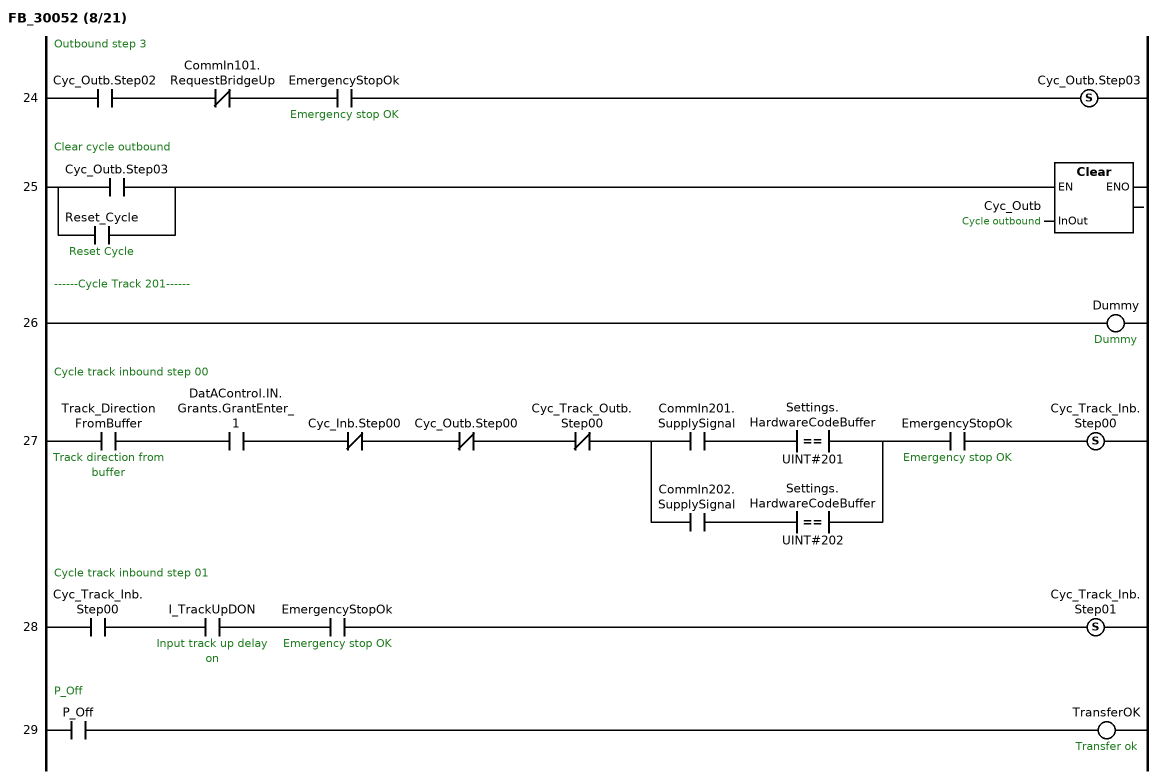
(* [picture p246: FB_30052, rungs 24-29] *)
(* Rung 24: Outbound step 3 *)
IF Cyc_Outb.Step02 AND NOT CommIn101.RequestBridgeUp AND EmergencyStopOk THEN
    Cyc_Outb.Step03 := TRUE;
END_IF;
(* Rung 25: Clear cycle outbound *)
IF Cyc_Outb.Step03 OR Reset_Cycle THEN Clear(InOut := Cyc_Outb); END_IF;
(* Rung 26: ------Cycle Track 201------ *)
Dummy := TRUE;
(* Rung 27: Cycle track inbound step 00 *)
IF Track_DirectionFromBuffer AND DatAControl.IN.Grants.GrantEnter_1 AND NOT Cyc_Inb.Step00 AND NOT Cyc_Outb.Step00 AND NOT Cyc_Track_Outb.Step00 AND ((CommIn201.SupplySignal AND (Settings.HardwareCodeBuffer = UINT#201)) OR (CommIn202.SupplySignal AND (Settings.HardwareCodeBuffer = UINT#202))) AND EmergencyStopOk THEN
    Cyc_Track_Inb.Step00 := TRUE;
END_IF;
(* Rung 28: Cycle track inbound step 01 *)
IF Cyc_Track_Inb.Step00 AND I_TrackUpDON AND EmergencyStopOk THEN Cyc_Track_Inb.Step01 := TRUE; END_IF;
(* Rung 29: P_Off *)
TransferOK := P_Off;

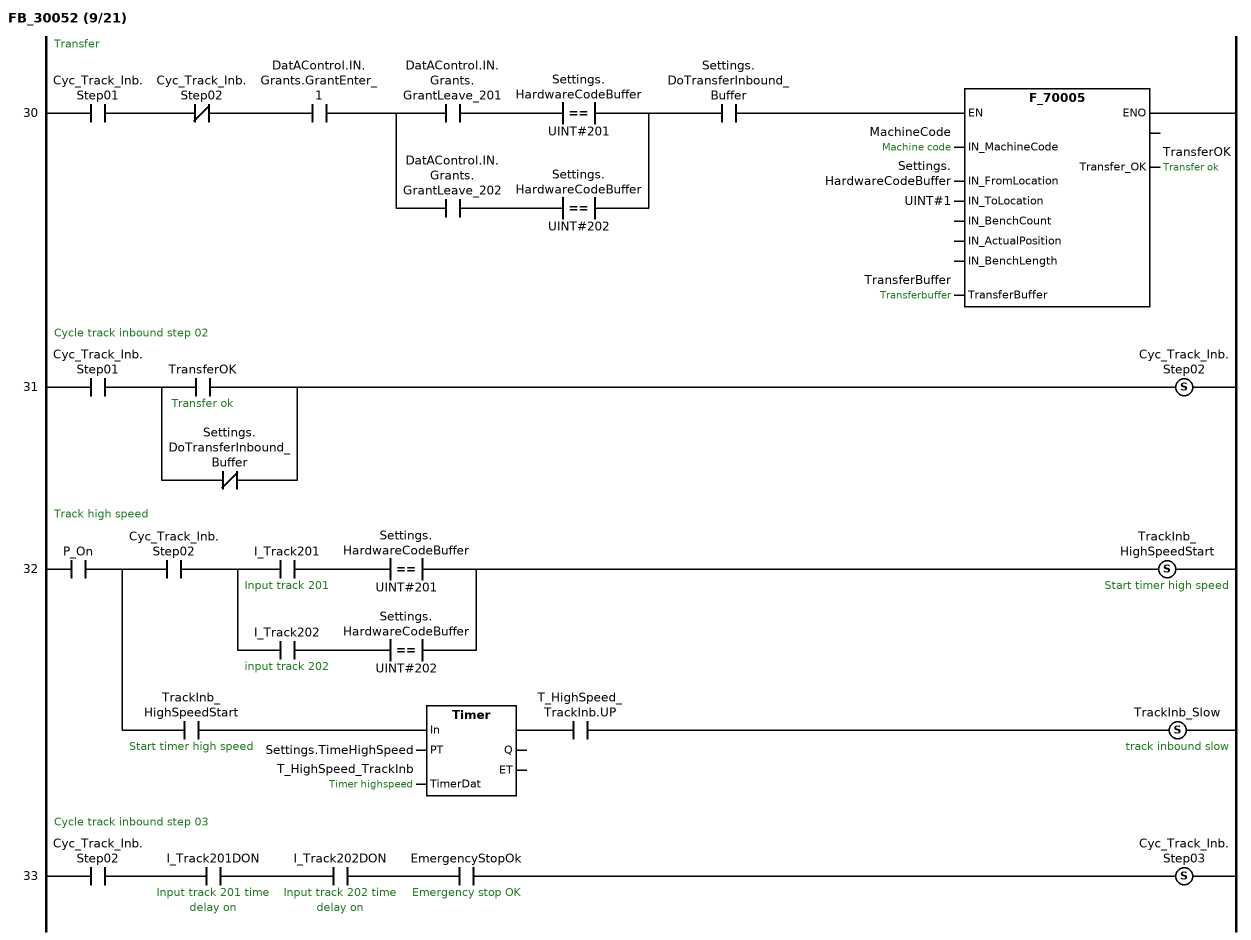
(* Rung 30: Transfer *)
IF Cyc_Track_Inb.Step01 AND NOT Cyc_Track_Inb.Step02 AND DatAControl.IN.Grants.GrantEnter_1 AND ((DatAControl.IN.Grants.GrantLeave_201 AND (Settings.HardwareCodeBuffer = UINT#201)) OR (DatAControl.IN.Grants.GrantLeave_202 AND (Settings.HardwareCodeBuffer = UINT#202))) AND Settings.DoTransferInbound_Buffer THEN
    F_70005(IN_MachineCode := MachineCode, IN_FromLocation := Settings.HardwareCodeBuffer, IN_ToLocation := UINT#1, TransferBuffer := TransferBuffer, Transfer_OK => TransferOK);
END_IF;
(* Rung 31: Cycle track inbound step 02 *)
IF Cyc_Track_Inb.Step01 AND (TransferOK OR NOT Settings.DoTransferInbound_Buffer) THEN
    Cyc_Track_Inb.Step02 := TRUE;
END_IF;
(* Rung 32: Track high speed *)
IF P_On AND Cyc_Track_Inb.Step02 AND ((I_Track201 AND (Settings.HardwareCodeBuffer = UINT#201)) OR (I_Track202 AND (Settings.HardwareCodeBuffer = UINT#202))) THEN
    TrackInb_HighSpeedStart := TRUE;
END_IF;
_t2 := Timer(In := P_On AND TrackInb_HighSpeedStart, PT := Settings.TimeHighSpeed, TimerDat := T_HighSpeed_TrackInb);
IF _t2 AND T_HighSpeed_TrackInb.UP THEN TrackInb_Slow := TRUE; END_IF;
(* Rung 33: Cycle track inbound step 03 *)
IF Cyc_Track_Inb.Step02 AND I_Track201DON AND I_Track202DON AND EmergencyStopOk THEN
    Cyc_Track_Inb.Step03 := TRUE;
END_IF;

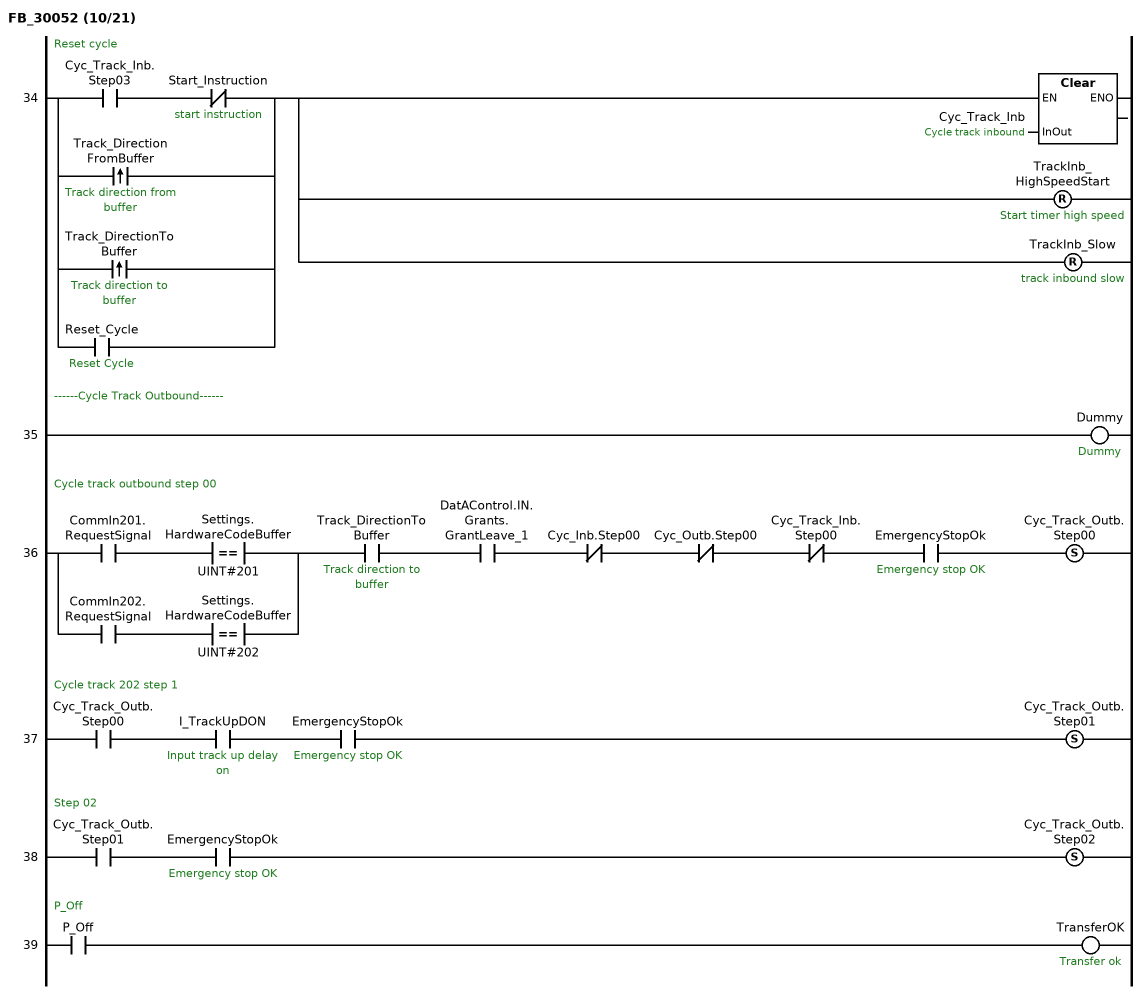
(* Rung 34: Reset cycle *)
_e3(CLK := Track_DirectionFromBuffer);
_e4(CLK := Track_DirectionToBuffer);
_p5 := (Cyc_Track_Inb.Step03 AND NOT Start_Instruction) OR _e3.Q OR _e4.Q OR Reset_Cycle;
IF _p5 THEN
    Clear(InOut := Cyc_Track_Inb);
    TrackInb_HighSpeedStart := FALSE;
    TrackInb_Slow := FALSE;
END_IF;
(* Rung 35: ------Cycle Track Outbound------ *)
Dummy := TRUE;
(* Rung 36: Cycle track outbound step 00 *)
IF ((CommIn201.RequestSignal AND (Settings.HardwareCodeBuffer = UINT#201)) OR (CommIn202.RequestSignal AND (Settings.HardwareCodeBuffer = UINT#202))) AND Track_DirectionToBuffer AND DatAControl.IN.Grants.GrantLeave_1 AND NOT Cyc_Inb.Step00 AND NOT Cyc_Outb.Step00 AND NOT Cyc_Track_Inb.Step00 AND EmergencyStopOk THEN
    Cyc_Track_Outb.Step00 := TRUE;
END_IF;
(* Rung 37: Cycle track 202 step 1 *)
IF Cyc_Track_Outb.Step00 AND I_TrackUpDON AND EmergencyStopOk THEN Cyc_Track_Outb.Step01 := TRUE; END_IF;
(* Rung 38: Step 02 *)
IF Cyc_Track_Outb.Step01 AND EmergencyStopOk THEN Cyc_Track_Outb.Step02 := TRUE; END_IF;
(* Rung 39: P_Off *)
TransferOK := P_Off;

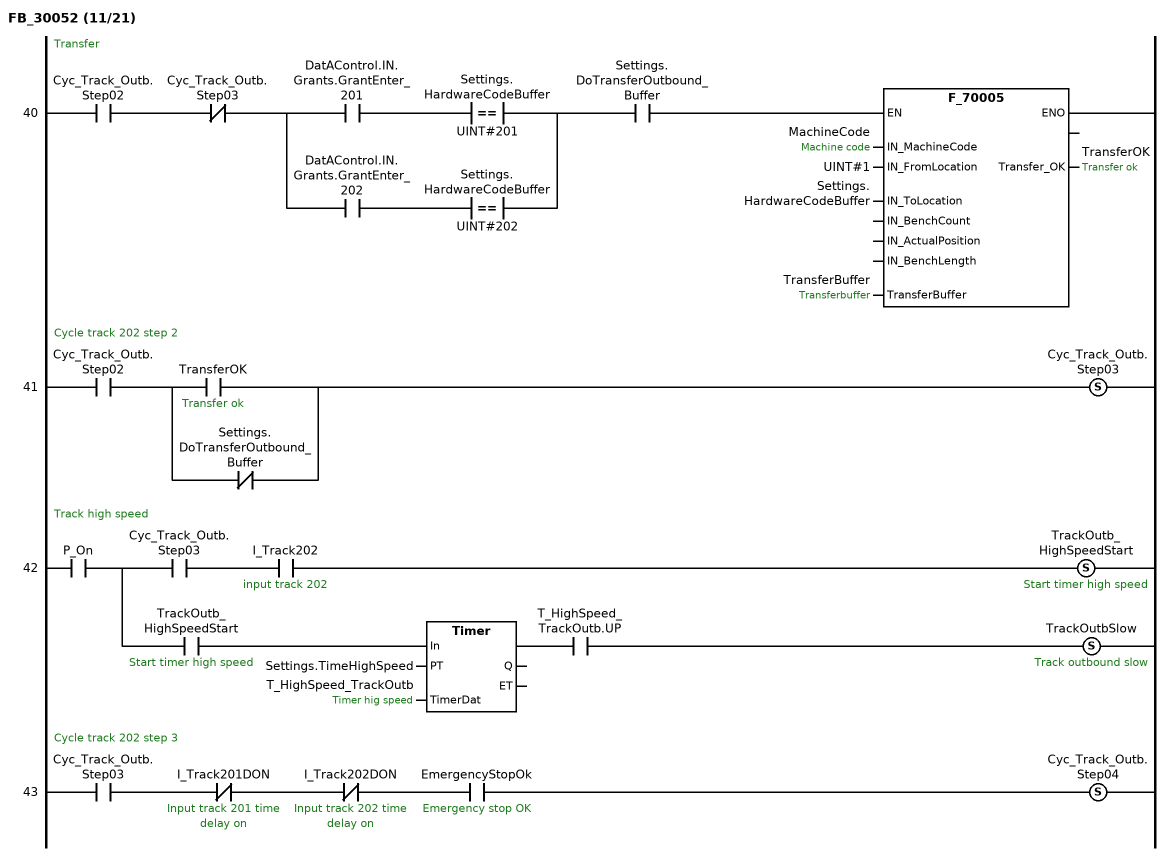
(* Rung 40: Transfer *)
IF Cyc_Track_Outb.Step02 AND NOT Cyc_Track_Outb.Step03 AND ((DatAControl.IN.Grants.GrantEnter_201 AND (Settings.HardwareCodeBuffer = UINT#201)) OR (DatAControl.IN.Grants.GrantEnter_202 AND (Settings.HardwareCodeBuffer = UINT#202))) AND Settings.DoTransferOutbound_Buffer THEN
    F_70005(IN_MachineCode := MachineCode, IN_FromLocation := UINT#1, IN_ToLocation := Settings.HardwareCodeBuffer, TransferBuffer := TransferBuffer, Transfer_OK => TransferOK);
END_IF;
(* Rung 41: Cycle track 202 step 2 *)
IF Cyc_Track_Outb.Step02 AND (TransferOK OR NOT Settings.DoTransferOutbound_Buffer) THEN
    Cyc_Track_Outb.Step03 := TRUE;
END_IF;
(* Rung 42: Track high speed *)
IF P_On AND Cyc_Track_Outb.Step03 AND I_Track202 THEN TrackOutb_HighSpeedStart := TRUE; END_IF;
_t6 := Timer(In := P_On AND TrackOutb_HighSpeedStart, PT := Settings.TimeHighSpeed, TimerDat := T_HighSpeed_TrackOutb);
IF _t6 AND T_HighSpeed_TrackOutb.UP THEN TrackOutbSlow := TRUE; END_IF;
(* Rung 43: Cycle track 202 step 3 *)
IF Cyc_Track_Outb.Step03 AND NOT I_Track201DON AND NOT I_Track202DON AND EmergencyStopOk THEN
    Cyc_Track_Outb.Step04 := TRUE;
END_IF;

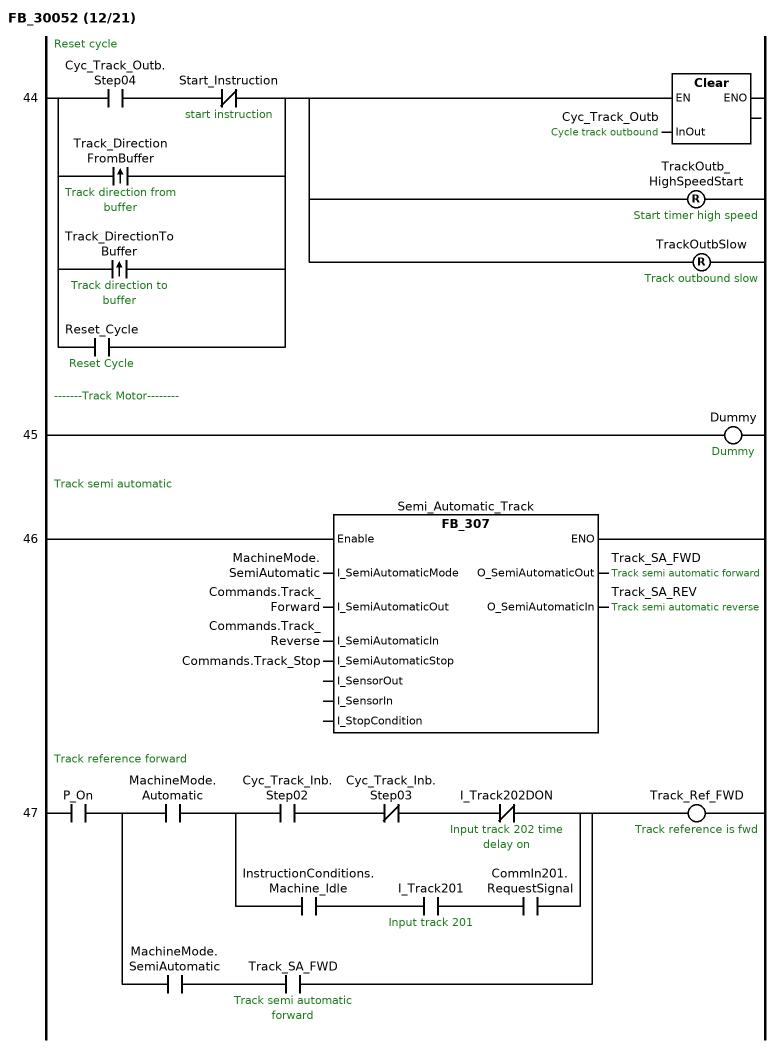
(* Rung 44: Reset cycle *)
_e7(CLK := Track_DirectionFromBuffer);
_e8(CLK := Track_DirectionToBuffer);
_p9 := (Cyc_Track_Outb.Step04 AND NOT Start_Instruction) OR _e7.Q OR _e8.Q OR Reset_Cycle;
IF _p9 THEN
    Clear(InOut := Cyc_Track_Outb);
    TrackOutb_HighSpeedStart := FALSE;
    TrackOutbSlow := FALSE;
END_IF;
(* Rung 45: -------Track Motor-------- *)
Dummy := TRUE;
(* Rung 46: Track semi automatic *)
Semi_Automatic_Track(Enable := TRUE, I_SemiAutomaticMode := MachineMode.SemiAutomatic, I_SemiAutomaticOut := Commands.Track_Forward, I_SemiAutomaticIn := Commands.Track_Reverse, I_SemiAutomaticStop := Commands.Track_Stop, O_SemiAutomaticOut => Track_SA_FWD, O_SemiAutomaticIn => Track_SA_REV);
(* Rung 47: Track reference forward *)
Track_Ref_FWD := P_On AND ((MachineMode.Automatic AND ((Cyc_Track_Inb.Step02 AND NOT Cyc_Track_Inb.Step03 AND NOT I_Track202DON) OR (InstructionConditions.Machine_Idle AND I_Track201 AND CommIn201.RequestSignal))) OR (MachineMode.SemiAutomatic AND Track_SA_FWD));

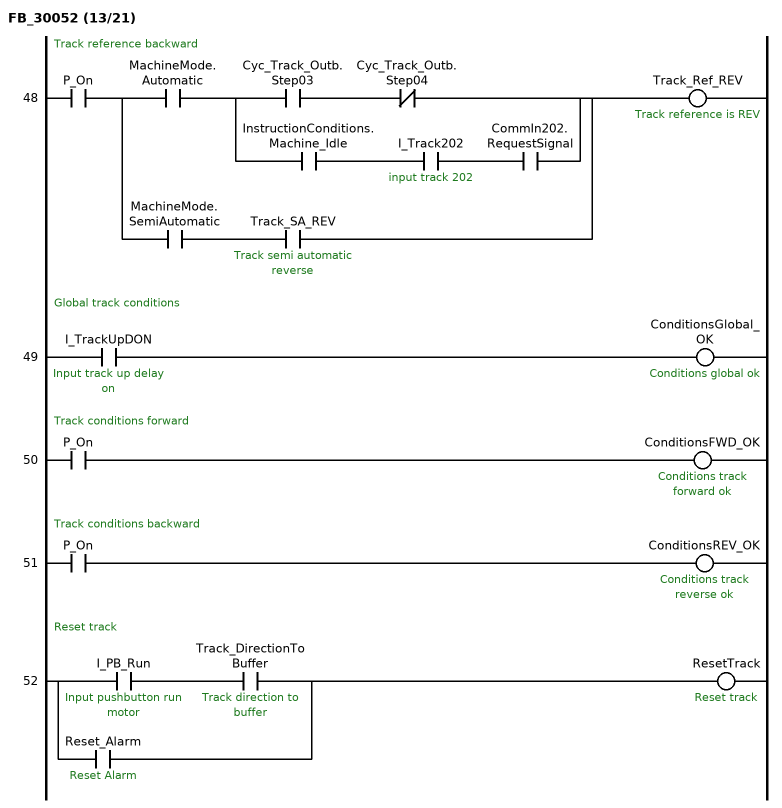
(* Rung 48: Track reference backward *)
Track_Ref_REV := P_On AND ((MachineMode.Automatic AND ((Cyc_Track_Outb.Step03 AND NOT Cyc_Track_Outb.Step04) OR (InstructionConditions.Machine_Idle AND I_Track202 AND CommIn202.RequestSignal))) OR (MachineMode.SemiAutomatic AND Track_SA_REV));
(* Rung 49: Global track conditions *)
ConditionsGlobal_OK := I_TrackUpDON;
(* Rung 50: Track conditions forward *)
ConditionsFWD_OK := P_On;
(* Rung 51: Track conditions backward *)
ConditionsREV_OK := P_On;
(* Rung 52: Reset track *)
ResetTrack := (I_PB_Run AND Track_DirectionToBuffer) OR Reset_Alarm;

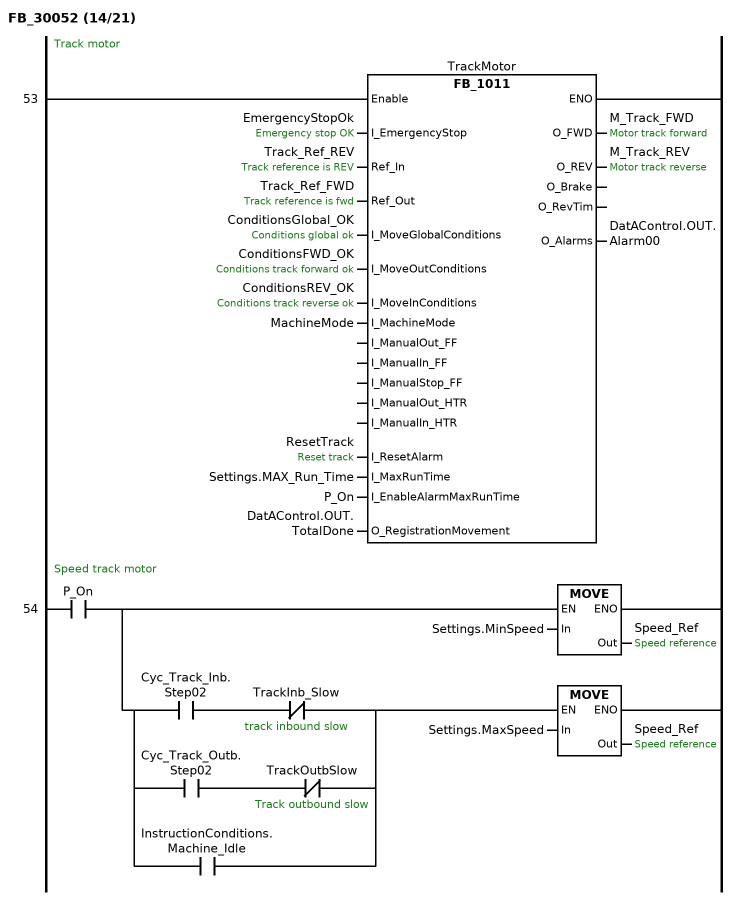
(* Rung 53: Track motor *)
TrackMotor(Enable := TRUE, I_EmergencyStop := EmergencyStopOk, Ref_In := Track_Ref_REV, Ref_Out := Track_Ref_FWD, I_MoveGlobalConditions := ConditionsGlobal_OK, I_MoveOutConditions := ConditionsFWD_OK, I_MoveInConditions := ConditionsREV_OK, I_MachineMode := MachineMode, I_ResetAlarm := ResetTrack, I_MaxRunTime := Settings.MAX_Run_Time, I_EnableAlarmMaxRunTime := P_On, O_RegistrationMovement := DatAControl.OUT.TotalDone, O_FWD => M_Track_FWD, O_REV => M_Track_REV, O_Alarms => DatAControl.OUT.Alarm00);
(* Rung 54: Speed track motor *)
IF P_On THEN Speed_Ref := Settings.MinSpeed; END_IF;
IF P_On AND ((Cyc_Track_Inb.Step02 AND NOT TrackInb_Slow) OR (Cyc_Track_Outb.Step02 AND NOT TrackOutbSlow) OR InstructionConditions.Machine_Idle) THEN
    Speed_Ref := Settings.MaxSpeed;
END_IF;

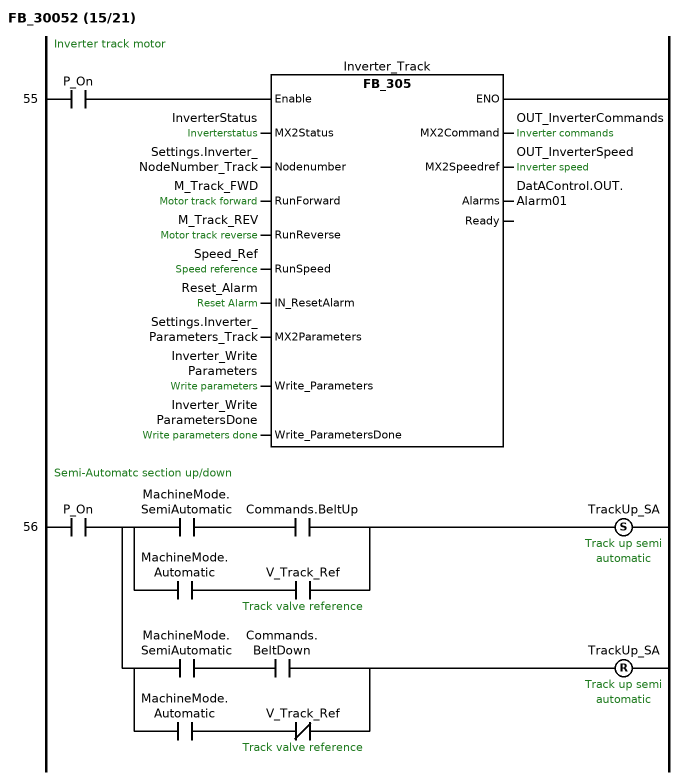
(* Rung 55: Inverter track motor *)
Inverter_Track(Enable := P_On, MX2Status := InverterStatus, Nodenumber := Settings.Inverter_NodeNumber_Track, RunForward := M_Track_FWD, RunReverse := M_Track_REV, RunSpeed := Speed_Ref, IN_ResetAlarm := Reset_Alarm, MX2Parameters := Settings.Inverter_Parameters_Track, Write_Parameters := Inverter_WriteParameters, Write_ParametersDone := Inverter_WriteParametersDone, MX2Command => OUT_InverterCommands, MX2Speedref => OUT_InverterSpeed, Alarms => DatAControl.OUT.Alarm01);
(* Rung 56: Semi-Automatc section up/down *)
IF P_On AND ((MachineMode.SemiAutomatic AND Commands.BeltUp) OR (MachineMode.Automatic AND V_Track_Ref)) THEN
    TrackUp_SA := TRUE;
END_IF;
IF P_On AND ((MachineMode.SemiAutomatic AND Commands.BeltDown) OR (MachineMode.Automatic AND NOT V_Track_Ref)) THEN
    TrackUp_SA := FALSE;
END_IF;

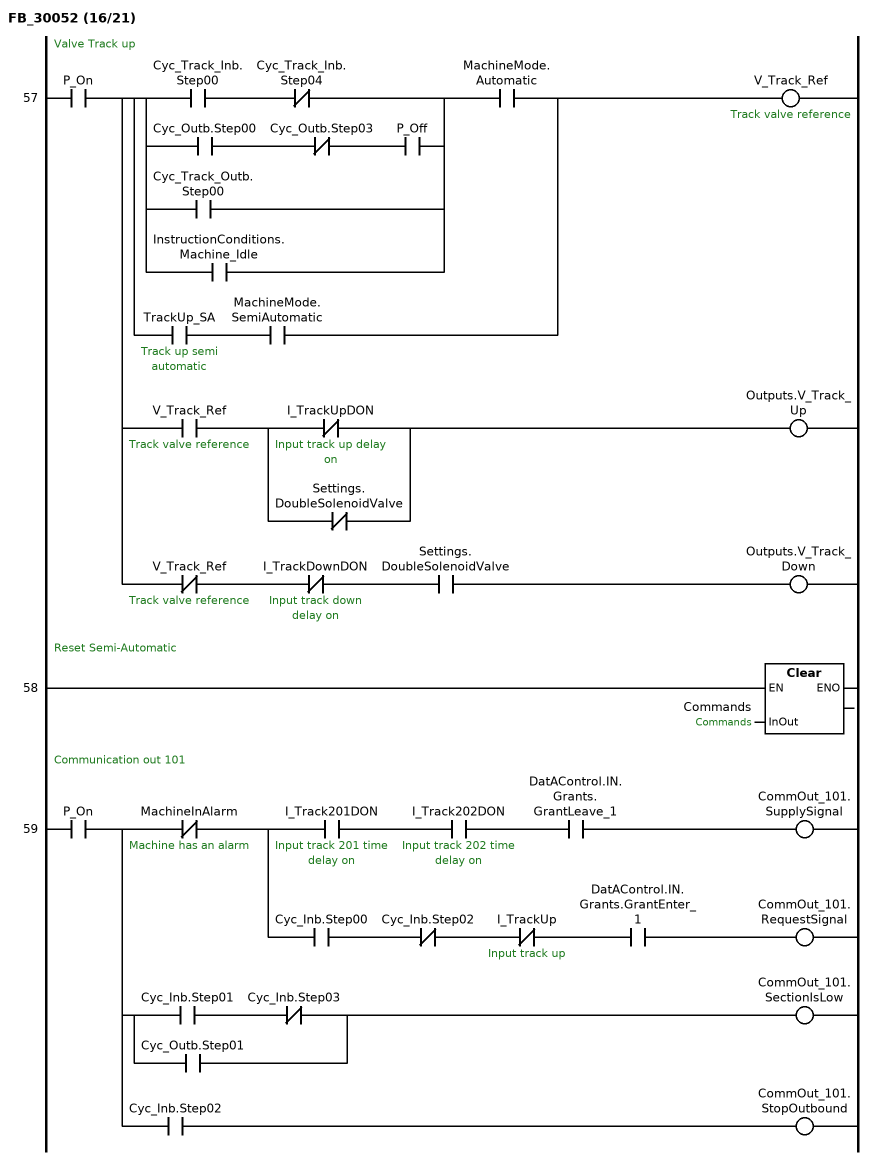
(* Rung 57: Valve Track up *)
V_Track_Ref := P_On AND ((((Cyc_Track_Inb.Step00 AND NOT Cyc_Track_Inb.Step04) OR (Cyc_Outb.Step00 AND NOT Cyc_Outb.Step03 AND P_Off) OR Cyc_Track_Outb.Step00 OR InstructionConditions.Machine_Idle) AND MachineMode.Automatic) OR (TrackUp_SA AND MachineMode.SemiAutomatic));
Outputs.V_Track_Up := P_On AND V_Track_Ref AND (NOT I_TrackUpDON OR NOT Settings.DoubleSolenoidValve);
Outputs.V_Track_Down := P_On AND NOT V_Track_Ref AND NOT I_TrackDownDON AND Settings.DoubleSolenoidValve;
(* Rung 58: Reset Semi-Automatic *)
Clear(InOut := Commands);
(* Rung 59: Communication out 101 *)
CommOut_101.SupplySignal := P_On AND NOT MachineInAlarm AND I_Track201DON AND I_Track202DON AND DatAControl.IN.Grants.GrantLeave_1;
CommOut_101.RequestSignal := P_On AND NOT MachineInAlarm AND Cyc_Inb.Step00 AND NOT Cyc_Inb.Step02 AND NOT I_TrackUp AND DatAControl.IN.Grants.GrantEnter_1;
CommOut_101.SectionIsLow := P_On AND ((Cyc_Inb.Step01 AND NOT Cyc_Inb.Step03) OR Cyc_Outb.Step01);
CommOut_101.StopOutbound := P_On AND Cyc_Inb.Step02;

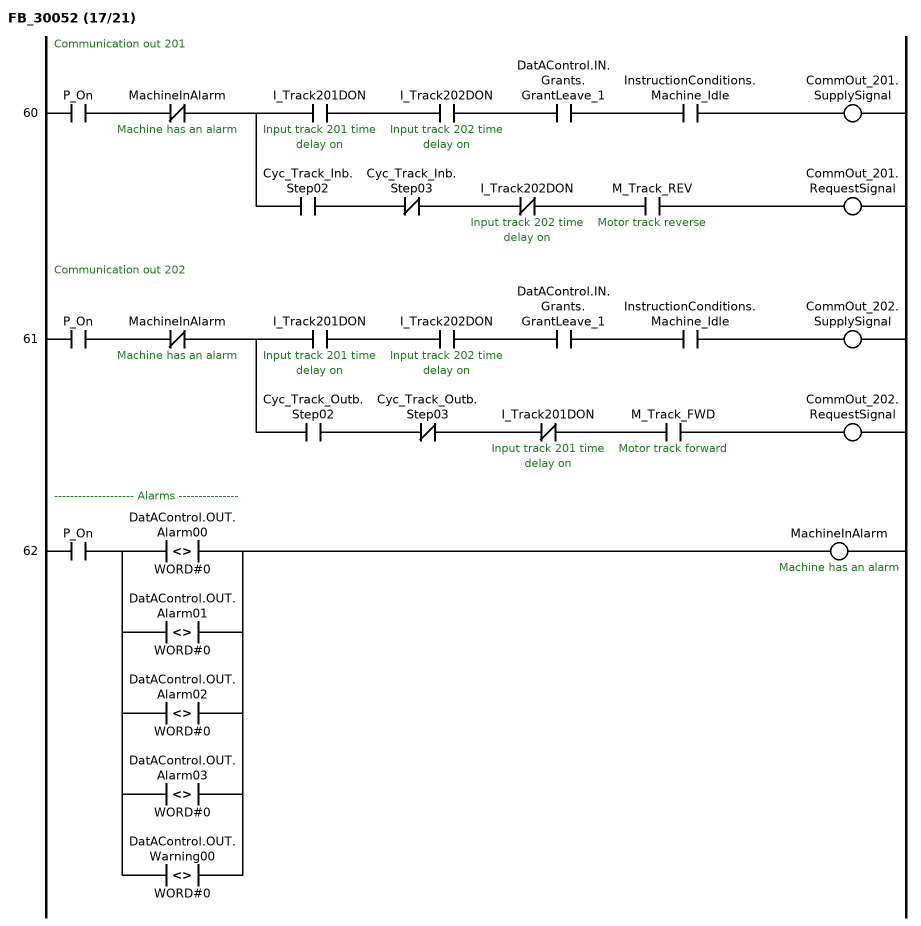
(* Rung 60: Communication out 201 *)
CommOut_201.SupplySignal := P_On AND NOT MachineInAlarm AND I_Track201DON AND I_Track202DON AND DatAControl.IN.Grants.GrantLeave_1 AND InstructionConditions.Machine_Idle;
CommOut_201.RequestSignal := P_On AND NOT MachineInAlarm AND Cyc_Track_Inb.Step02 AND NOT Cyc_Track_Inb.Step03 AND NOT I_Track202DON AND M_Track_REV;
(* Rung 61: Communication out 202 *)
CommOut_202.SupplySignal := P_On AND NOT MachineInAlarm AND I_Track201DON AND I_Track202DON AND DatAControl.IN.Grants.GrantLeave_1 AND InstructionConditions.Machine_Idle;
CommOut_202.RequestSignal := P_On AND NOT MachineInAlarm AND Cyc_Track_Outb.Step02 AND NOT Cyc_Track_Outb.Step03 AND NOT I_Track201DON AND M_Track_FWD;
(* Rung 62: -------------------- Alarms --------------- *)
MachineInAlarm := P_On AND ((DatAControl.OUT.Alarm00 <> WORD#0) OR (DatAControl.OUT.Alarm01 <> WORD#0) OR (DatAControl.OUT.Alarm02 <> WORD#0) OR (DatAControl.OUT.Alarm03 <> WORD#0) OR (DatAControl.OUT.Warning00 <> WORD#0));

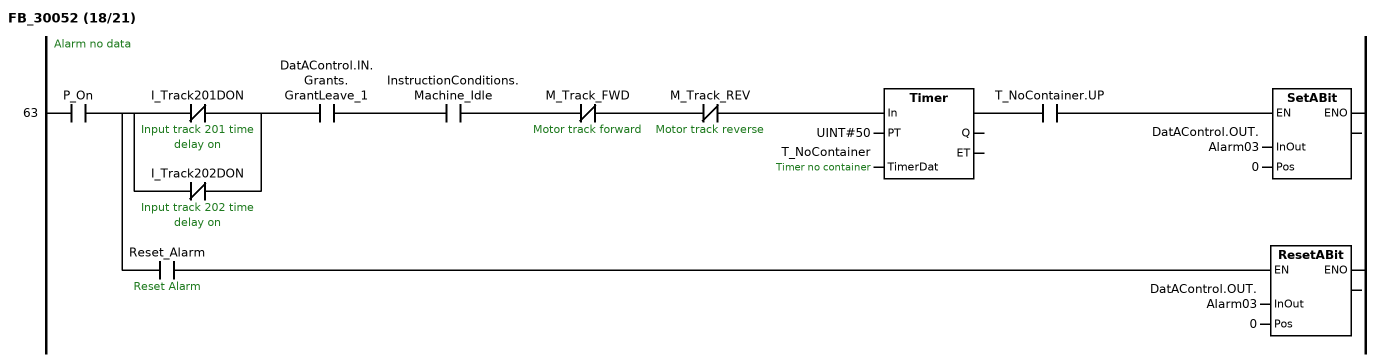
(* Rung 63: Alarm no data *)
_t10 := Timer(In := P_On AND (NOT I_Track201DON OR NOT I_Track202DON) AND DatAControl.IN.Grants.GrantLeave_1 AND InstructionConditions.Machine_Idle AND NOT M_Track_FWD AND NOT M_Track_REV, PT := UINT#50, TimerDat := T_NoContainer);
IF _t10 AND T_NoContainer.UP THEN SetABit(InOut := DatAControl.OUT.Alarm03, Pos := 0); END_IF;
IF P_On AND Reset_Alarm THEN ResetABit(InOut := DatAControl.OUT.Alarm03, Pos := 0); END_IF;

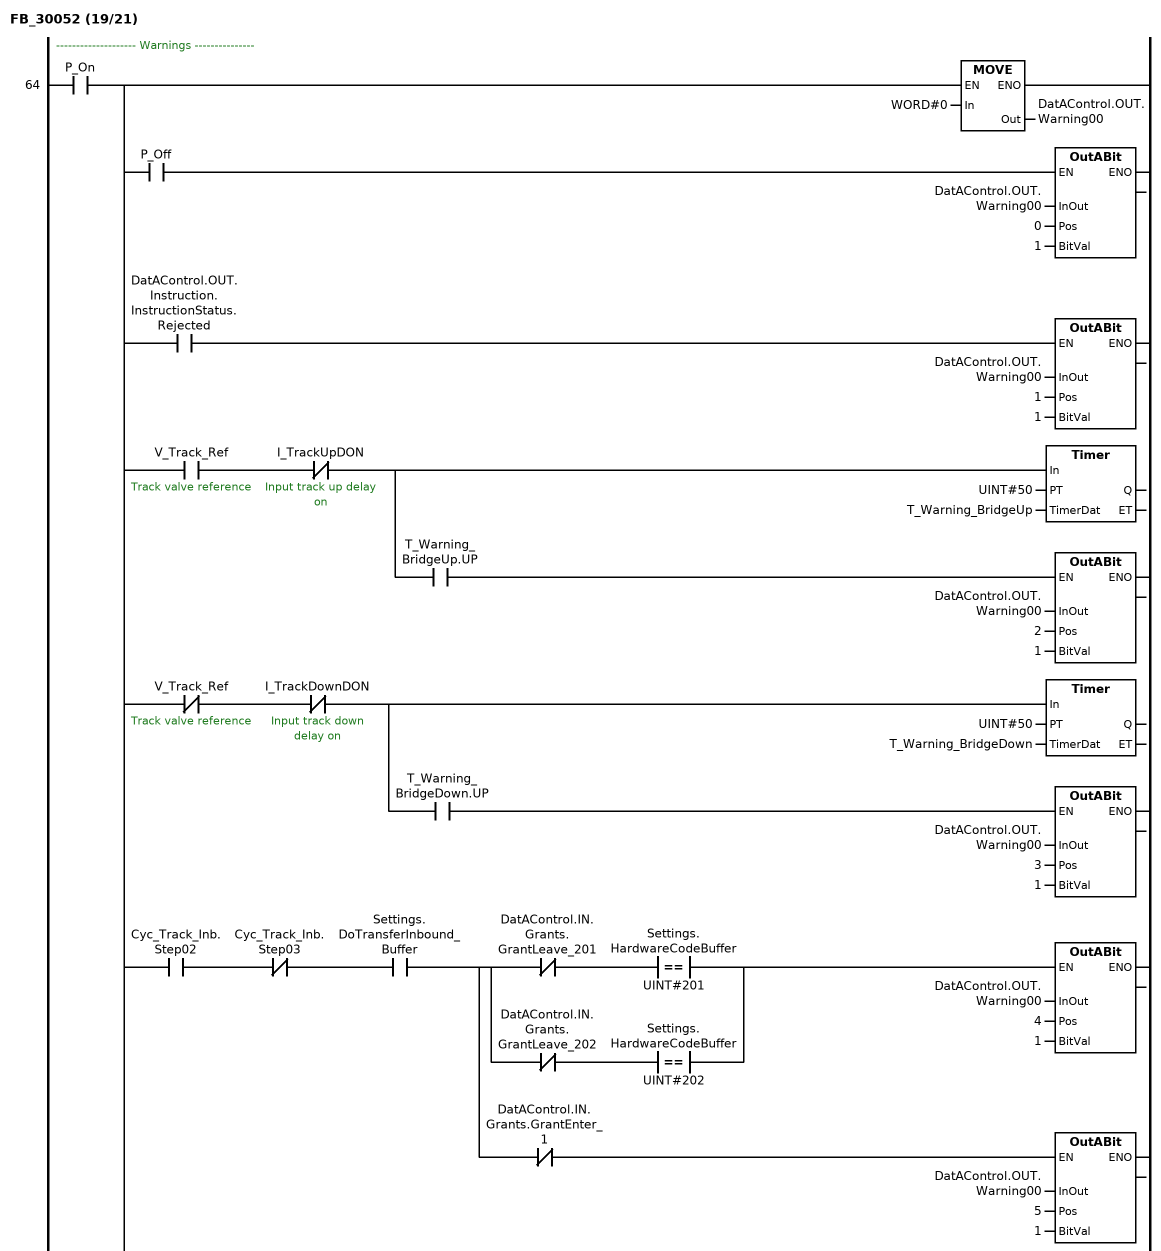

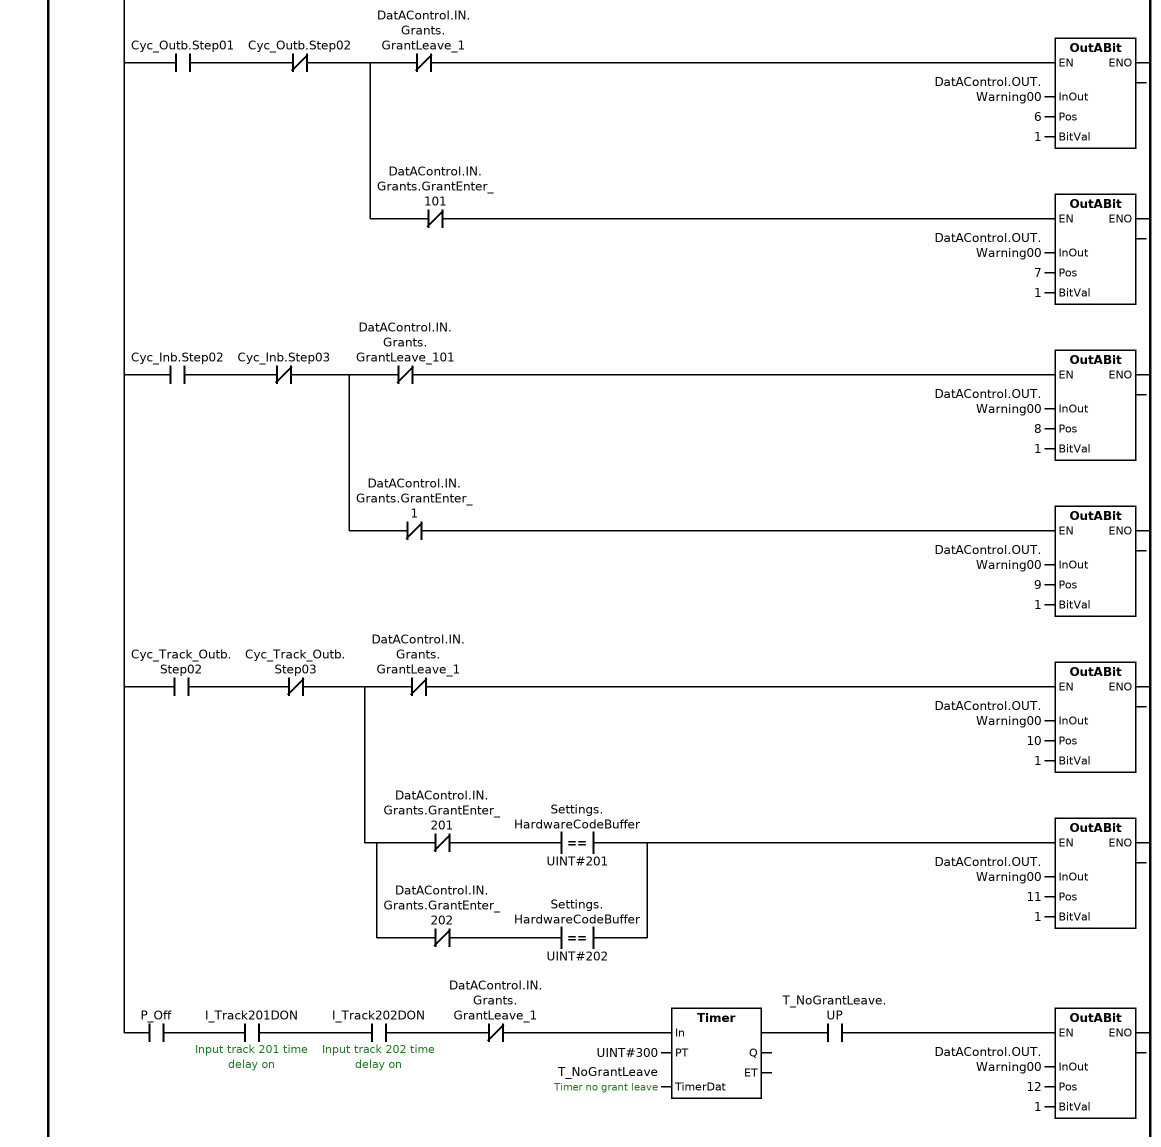
(* Rung 64: -------------------- Warnings --------------- *)
IF P_On THEN DatAControl.OUT.Warning00 := WORD#0; END_IF;
IF P_On AND P_Off THEN OutABit(InOut := DatAControl.OUT.Warning00, Pos := 0, BitVal := 1); END_IF;
IF P_On AND DatAControl.OUT.Instruction.InstructionStatus.Rejected THEN
    OutABit(InOut := DatAControl.OUT.Warning00, Pos := 1, BitVal := 1);
END_IF;
_t11 := Timer(In := P_On AND V_Track_Ref AND NOT I_TrackUpDON, PT := UINT#50, TimerDat := T_Warning_BridgeUp);
IF P_On AND V_Track_Ref AND NOT I_TrackUpDON AND T_Warning_BridgeUp.UP THEN
    OutABit(InOut := DatAControl.OUT.Warning00, Pos := 2, BitVal := 1);
END_IF;
_t12 := Timer(In := P_On AND NOT V_Track_Ref AND NOT I_TrackDownDON, PT := UINT#50, TimerDat := T_Warning_BridgeDown);
IF P_On AND NOT V_Track_Ref AND NOT I_TrackDownDON AND T_Warning_BridgeDown.UP THEN
    OutABit(InOut := DatAControl.OUT.Warning00, Pos := 3, BitVal := 1);
END_IF;
_p13 := P_On AND Cyc_Track_Inb.Step02 AND NOT Cyc_Track_Inb.Step03 AND Settings.DoTransferInbound_Buffer;
IF _p13 AND ((NOT DatAControl.IN.Grants.GrantLeave_201 AND (Settings.HardwareCodeBuffer = UINT#201)) OR (NOT DatAControl.IN.Grants.GrantLeave_202 AND (Settings.HardwareCodeBuffer = UINT#202))) THEN
    OutABit(InOut := DatAControl.OUT.Warning00, Pos := 4, BitVal := 1);
END_IF;
IF _p13 AND NOT DatAControl.IN.Grants.GrantEnter_1 THEN
    OutABit(InOut := DatAControl.OUT.Warning00, Pos := 5, BitVal := 1);
END_IF;
IF P_On AND Cyc_Outb.Step01 AND NOT Cyc_Outb.Step02 AND NOT DatAControl.IN.Grants.GrantLeave_1 THEN
    OutABit(InOut := DatAControl.OUT.Warning00, Pos := 6, BitVal := 1);
END_IF;
IF P_On AND Cyc_Outb.Step01 AND NOT Cyc_Outb.Step02 AND NOT DatAControl.IN.Grants.GrantEnter_101 THEN
    OutABit(InOut := DatAControl.OUT.Warning00, Pos := 7, BitVal := 1);
END_IF;
IF P_On AND Cyc_Inb.Step02 AND NOT Cyc_Inb.Step03 AND NOT DatAControl.IN.Grants.GrantLeave_101 THEN
    OutABit(InOut := DatAControl.OUT.Warning00, Pos := 8, BitVal := 1);
END_IF;
IF P_On AND Cyc_Inb.Step02 AND NOT Cyc_Inb.Step03 AND NOT DatAControl.IN.Grants.GrantEnter_1 THEN
    OutABit(InOut := DatAControl.OUT.Warning00, Pos := 9, BitVal := 1);
END_IF;
_p14 := P_On AND Cyc_Track_Outb.Step02 AND NOT Cyc_Track_Outb.Step03;
IF _p14 AND NOT DatAControl.IN.Grants.GrantLeave_1 THEN
    OutABit(InOut := DatAControl.OUT.Warning00, Pos := 10, BitVal := 1);
END_IF;
IF _p14 AND ((NOT DatAControl.IN.Grants.GrantEnter_201 AND (Settings.HardwareCodeBuffer = UINT#201)) OR (NOT DatAControl.IN.Grants.GrantEnter_202 AND (Settings.HardwareCodeBuffer = UINT#202))) THEN
    OutABit(InOut := DatAControl.OUT.Warning00, Pos := 11, BitVal := 1);
END_IF;
_t15 := Timer(In := P_On AND P_Off AND I_Track201DON AND I_Track202DON AND NOT DatAControl.IN.Grants.GrantLeave_1, PT := UINT#300, TimerDat := T_NoGrantLeave);
IF _t15 AND T_NoGrantLeave.UP THEN
    OutABit(InOut := DatAControl.OUT.Warning00, Pos := 12, BitVal := 1);
END_IF;

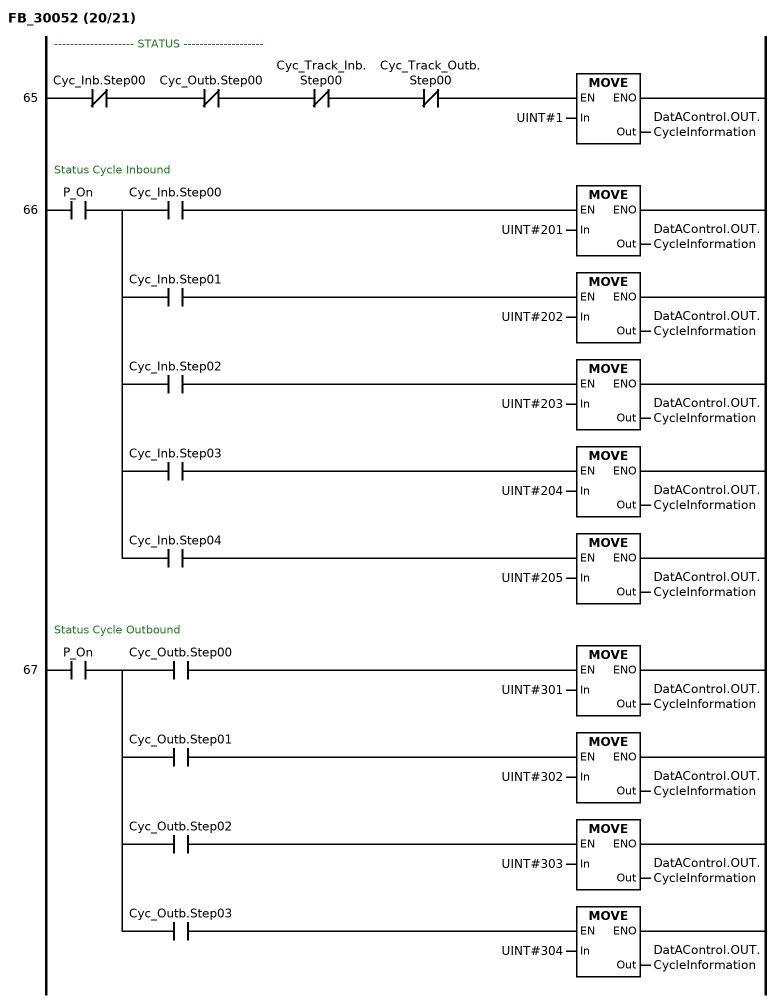
(* Rung 65: -------------------- STATUS -------------------- *)
IF NOT Cyc_Inb.Step00 AND NOT Cyc_Outb.Step00 AND NOT Cyc_Track_Inb.Step00 AND NOT Cyc_Track_Outb.Step00 THEN
    DatAControl.OUT.CycleInformation := UINT#1;
END_IF;
(* Rung 66: Status Cycle Inbound *)
IF P_On AND Cyc_Inb.Step00 THEN DatAControl.OUT.CycleInformation := UINT#201; END_IF;
IF P_On AND Cyc_Inb.Step01 THEN DatAControl.OUT.CycleInformation := UINT#202; END_IF;
IF P_On AND Cyc_Inb.Step02 THEN DatAControl.OUT.CycleInformation := UINT#203; END_IF;
IF P_On AND Cyc_Inb.Step03 THEN DatAControl.OUT.CycleInformation := UINT#204; END_IF;
IF P_On AND Cyc_Inb.Step04 THEN DatAControl.OUT.CycleInformation := UINT#205; END_IF;
(* Rung 67: Status Cycle Outbound *)
IF P_On AND Cyc_Outb.Step00 THEN DatAControl.OUT.CycleInformation := UINT#301; END_IF;
IF P_On AND Cyc_Outb.Step01 THEN DatAControl.OUT.CycleInformation := UINT#302; END_IF;
IF P_On AND Cyc_Outb.Step02 THEN DatAControl.OUT.CycleInformation := UINT#303; END_IF;
IF P_On AND Cyc_Outb.Step03 THEN DatAControl.OUT.CycleInformation := UINT#304; END_IF;

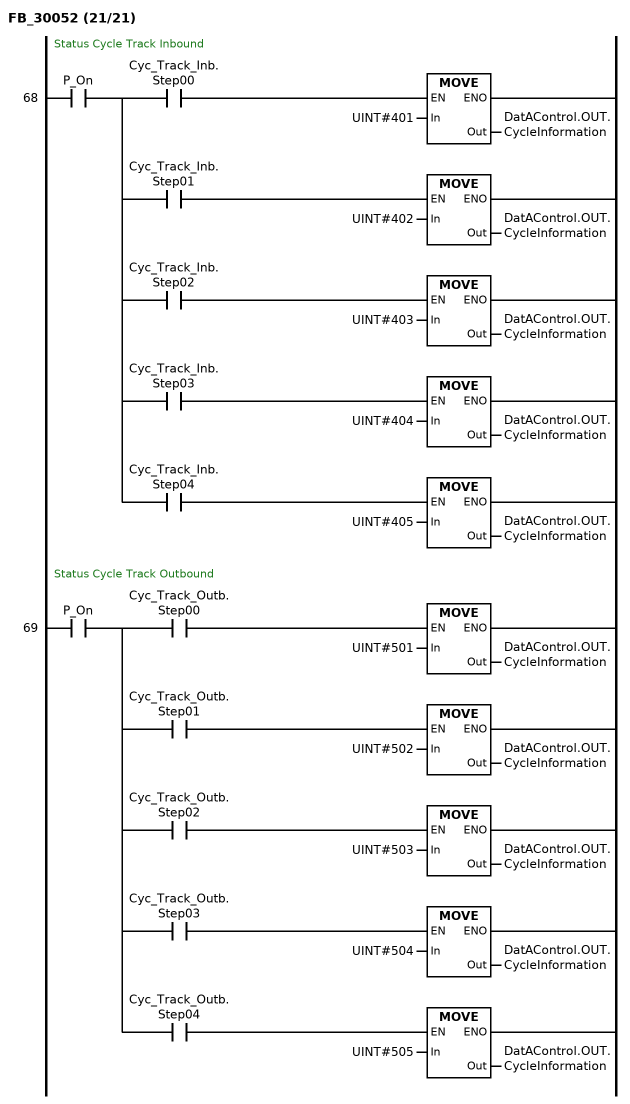
(* Rung 68: Status Cycle Track Inbound *)
IF P_On AND Cyc_Track_Inb.Step00 THEN DatAControl.OUT.CycleInformation := UINT#401; END_IF;
IF P_On AND Cyc_Track_Inb.Step01 THEN DatAControl.OUT.CycleInformation := UINT#402; END_IF;
IF P_On AND Cyc_Track_Inb.Step02 THEN DatAControl.OUT.CycleInformation := UINT#403; END_IF;
IF P_On AND Cyc_Track_Inb.Step03 THEN DatAControl.OUT.CycleInformation := UINT#404; END_IF;
IF P_On AND Cyc_Track_Inb.Step04 THEN DatAControl.OUT.CycleInformation := UINT#405; END_IF;
(* Rung 69: Status Cycle Track Outbound *)
IF P_On AND Cyc_Track_Outb.Step00 THEN DatAControl.OUT.CycleInformation := UINT#501; END_IF;
IF P_On AND Cyc_Track_Outb.Step01 THEN DatAControl.OUT.CycleInformation := UINT#502; END_IF;
IF P_On AND Cyc_Track_Outb.Step02 THEN DatAControl.OUT.CycleInformation := UINT#503; END_IF;
IF P_On AND Cyc_Track_Outb.Step03 THEN DatAControl.OUT.CycleInformation := UINT#504; END_IF;
IF P_On AND Cyc_Track_Outb.Step04 THEN DatAControl.OUT.CycleInformation := UINT#505; END_IF;
END_FUNCTION_BLOCK